FUNCTION_BLOCK PUBL_1 (* 2-variable data publisher *)
  (* Standard: 61499-2 *)
  (* Version 1.0, 21-03-12, GASR, Universidade do Estado de Santa Catarina *)
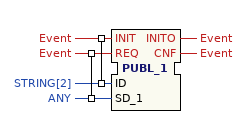
  EVENT_INPUT
    INIT WITH ID; (* Service initiaization *)
    REQ WITH SD_1;
  END_EVENT
  EVENT_OUTPUT
    INITO; (* Initialization Confirm *)
    CNF; (* Service confirmation *)
  END_EVENT
  VAR_INPUT
    ID : ARRAY [0..1] OF STRING; (* Default id is the FB instance name *)
    SD_1 : ANY;
  END_VAR
  SERVICE PUBL_105/SUBL_105 (* Data publication service *)
    SEQUENCE normal_establishment
      PUBL_105.INIT(ID) -> PUBL_105.INITO();
      SUBL_105.INIT(ID) -> SUBL_105.INITO();
    END_SEQUENCE
    SEQUENCE normal_data_transfer
      PUBL_105.REQ(SD_1) -> Subl_105.IND(RD_1);
    END_SEQUENCE
  END_SERVICE
END_FUNCTION_BLOCK
